(* PLC project process, Dassault Systèmes ControlBuild 2024x *)
(* stored: creationDateTime 2023-10-03T11:13:42-01:00 *)

PROGRAM bottling_line.process
  VAR_INPUT
    highLevel1 : BOOL := false;
    lowLevel1 : BOOL := false;
  END_VAR
  VAR_INPUT
    highLevel2 : BOOL := false;
    lowLevel2 : BOOL := false;
  END_VAR
  VAR_INPUT
    highLevel3 : BOOL := false;
    lowLevel3 : BOOL := false;
  END_VAR
  VAR_INPUT
    startCyclePB : BOOL := false;
    initPB : BOOL := false;
    preparationPB : BOOL := false;
    productionPB : BOOL := false;
    closingPB : BOOL := false;
  END_VAR
  VAR_INPUT
    pulseGenerator : BOOL := false;
    bottleFilled : BOOL := false;
    bottlePresent : BOOL := false;
  END_VAR
  VAR_OUTPUT
    load : BOOL := false;
    evacuate : BOOL := false;
    convoy : BOOL := false;
  END_VAR
  VAR_OUTPUT
    pump1 : BOOL := false;
    pump2 : BOOL := false;
    valve1 : BOOL := false;
    valve2 : BOOL := false;
    valve3 : BOOL := false;
    valve4 : BOOL := false;
    loSpeedAgitator : BOOL := false;
    hiSpeedAgitator : BOOL := false;
  END_VAR
  VAR_OUTPUT
    valve5 : BOOL := false;
  END_VAR

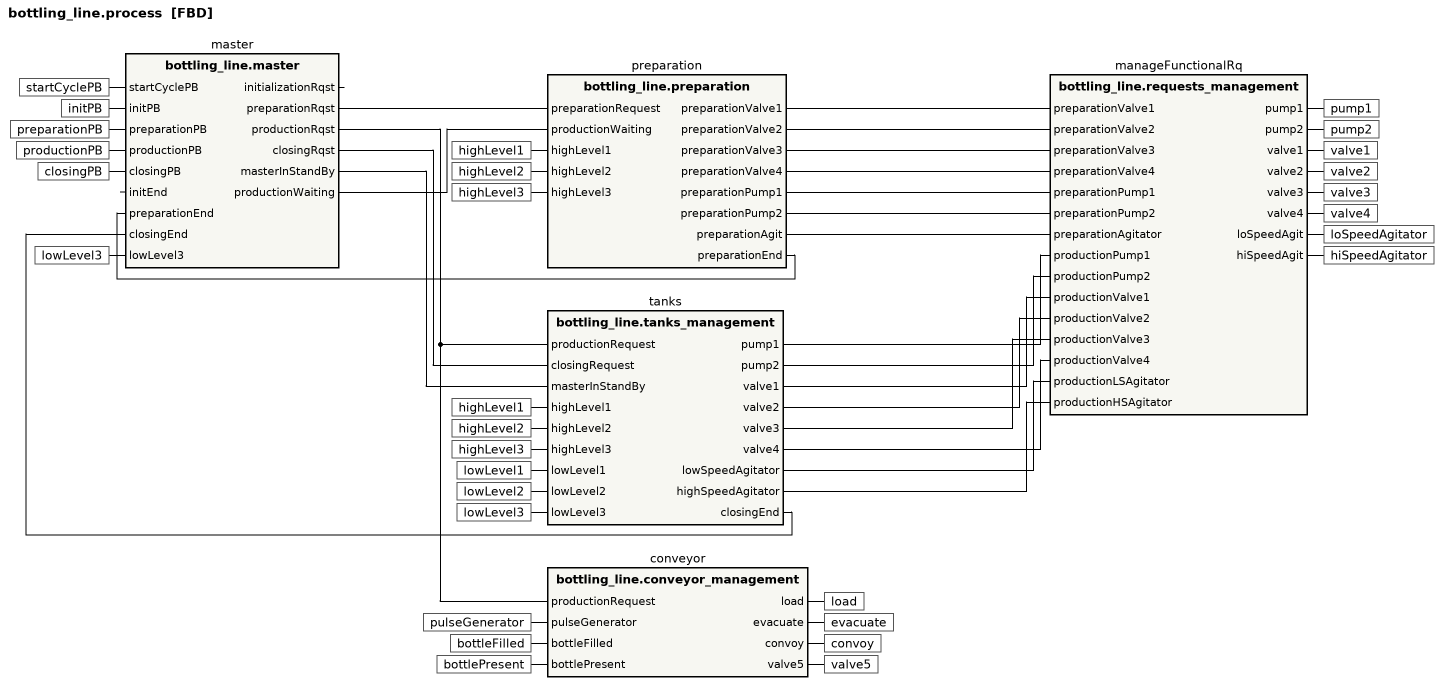
(* FBD diagram, written out as Structured Text *)
preparation(preparationRequest := master.preparationRqst, productionWaiting := master.productionWaiting, highLevel1 := highLevel1, highLevel2 := highLevel2, highLevel3 := highLevel3);
tanks(productionRequest := master.productionRqst, closingRequest := master.closingRqst, masterInStandBy := master.masterInStandBy, highLevel1 := highLevel1, highLevel2 := highLevel2, highLevel3 := highLevel3, lowLevel1 := lowLevel1, lowLevel2 := lowLevel2, lowLevel3 := lowLevel3);
master(startCyclePB := startCyclePB, initPB := initPB, preparationPB := preparationPB, productionPB := productionPB, closingPB := closingPB, preparationEnd := preparation.preparationEnd, closingEnd := tanks.closingEnd, lowLevel3 := lowLevel3);
conveyor(productionRequest := master.productionRqst, pulseGenerator := pulseGenerator, bottleFilled := bottleFilled, bottlePresent := bottlePresent);
load := conveyor.load;
evacuate := conveyor.evacuate;
convoy := conveyor.convoy;
valve5 := conveyor.valve5;
manageFunctionalRq(preparationValve1 := preparation.preparationValve1, preparationValve2 := preparation.preparationValve2, preparationValve3 := preparation.preparationValve3, preparationValve4 := preparation.preparationValve4, preparationPump1 := preparation.preparationPump1, preparationPump2 := preparation.preparationPump2, preparationAgitator := preparation.preparationAgit, productionPump1 := tanks.pump1, productionPump2 := tanks.pump2, productionValve1 := tanks.valve1, productionValve2 := tanks.valve2, productionValve3 := tanks.valve3, productionValve4 := tanks.valve4, productionLSAgitator := tanks.lowSpeedAgitator, productionHSAgitator := tanks.highSpeedAgitator);
pump1 := manageFunctionalRq.pump1;
pump2 := manageFunctionalRq.pump2;
valve1 := manageFunctionalRq.valve1;
valve2 := manageFunctionalRq.valve2;
valve3 := manageFunctionalRq.valve3;
valve4 := manageFunctionalRq.valve4;
loSpeedAgitator := manageFunctionalRq.loSpeedAgit;
hiSpeedAgitator := manageFunctionalRq.hiSpeedAgit;
END_PROGRAM
